FUNCTION_BLOCK NormallyOpenPushButton IMPLEMENTS I_PushButton
VAR
	input AT%I* : BOOL;
END_VAR

PROPERTY PUBLIC isPressed : BOOL
GET
isPressed	:=	input;
END_GET
END_PROPERTY

PROPERTY PUBLIC isReleased : BOOL
GET
isReleased	:=	NOT input;
END_GET
END_PROPERTY

END_FUNCTION_BLOCK

(* stored: Version 1.1.0.1, ProductVersion 3.1.4024.12
   POU NormallyOpenPushButton: Id {75854eaf-c318-4add-8e14-b5c5a74bb787}, SpecialFunc None
   Property isPressed: Id {573f6b29-ea29-4e82-8f11-d0b15dc9b262}
   Get Get: Id {5bc582f9-11a9-4f61-ba8c-26bda3f4d012}
   Property isReleased: Id {e89798a2-1a96-4659-9bec-2aa1df4a8dba}
   Get Get: Id {c479b94a-70fd-47db-b58a-840f79a50b55} *)
